SUBAPPLICATION Uebung_052_AX (* DigitalInput_I1-_I4 auf DigitalOutput_Q1-_Q4, mit Plug and Socket *)
  (* Standard: 61499-2; Description: Copyright (c) 2026 Meisterschulen am Ostbahnhof This program and the accompanying materials are made available under the terms of the Eclipse Public License 2.0 which is available at https://www.eclipse.org/legal/epl-2.0/ SPDX-License-Identifier: EPL-2.0 *)
  (* Version 1.0, 2026-09-09, Franz Höpfinger, Meisterschulen am Ostbahnhof, initial API and implementation and/or initial documentation *)
  PACKAGE Uebungen;
  IMPORT logiBUS::io::DI::logiBUS_DI::Input_I1;
  IMPORT logiBUS::io::DI::logiBUS_DI::Input_I2;
  IMPORT logiBUS::io::DI::logiBUS_DI::Input_I3;
  IMPORT logiBUS::io::DI::logiBUS_DI::Input_I4;
  IMPORT logiBUS::io::DQ::logiBUS_DO::Output_Q1;
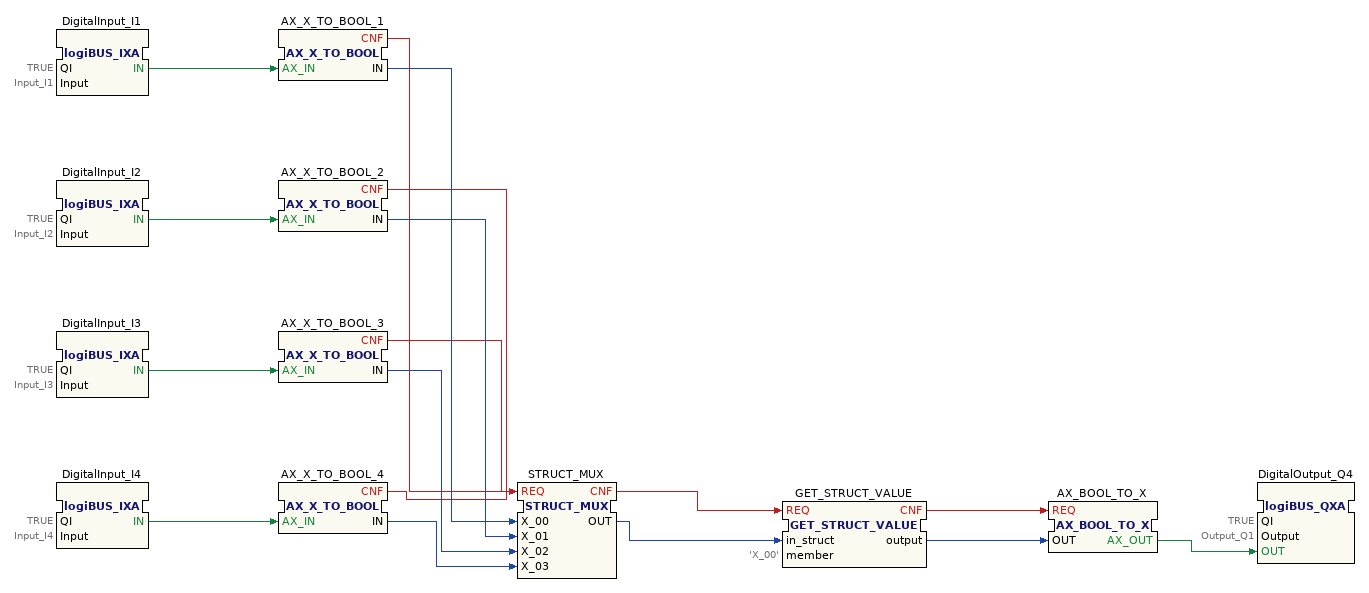
  FBS
    DigitalInput_I1 : logiBUS::io::DI::logiBUS_IXA(QI := TRUE, Input := Input_I1);
    DigitalInput_I2 : logiBUS::io::DI::logiBUS_IXA(QI := TRUE, Input := Input_I2);
    DigitalInput_I3 : logiBUS::io::DI::logiBUS_IXA(QI := TRUE, Input := Input_I3);
    DigitalOutput_Q4 : logiBUS::io::DQ::logiBUS_QXA(QI := TRUE, Output := Output_Q1);
    DigitalInput_I4 : logiBUS::io::DI::logiBUS_IXA(QI := TRUE, Input := Input_I4);
    GET_STRUCT_VALUE : eclipse4diac::convert::GET_STRUCT_VALUE(member := 'X_00');
    STRUCT_MUX : eclipse4diac::convert::STRUCT_MUX; {SET_ATTRIBUTE(StructuredType, logiBUS::utils::conversion::types::ST04X)}
    AX_X_TO_BOOL_1 : adapter::conversion::unidirectional::AX_X_TO_BOOL;
    AX_X_TO_BOOL_2 : adapter::conversion::unidirectional::AX_X_TO_BOOL;
    AX_X_TO_BOOL_3 : adapter::conversion::unidirectional::AX_X_TO_BOOL;
    AX_X_TO_BOOL_4 : adapter::conversion::unidirectional::AX_X_TO_BOOL;
    AX_BOOL_TO_X : adapter::conversion::unidirectional::AX_BOOL_TO_X;
  END_FBS
  EVENT_CONNECTIONS
    GET_STRUCT_VALUE.CNF TO AX_BOOL_TO_X.REQ;
    AX_X_TO_BOOL_1.CNF TO STRUCT_MUX.REQ;
    AX_X_TO_BOOL_2.CNF TO STRUCT_MUX.REQ;
    AX_X_TO_BOOL_3.CNF TO STRUCT_MUX.REQ;
    AX_X_TO_BOOL_4.CNF TO STRUCT_MUX.REQ;
    STRUCT_MUX.CNF TO GET_STRUCT_VALUE.REQ;
  END_CONNECTIONS
  DATA_CONNECTIONS
    GET_STRUCT_VALUE.output TO AX_BOOL_TO_X.OUT;
    AX_X_TO_BOOL_1.IN TO STRUCT_MUX.X_00;
    AX_X_TO_BOOL_2.IN TO STRUCT_MUX.X_01;
    AX_X_TO_BOOL_3.IN TO STRUCT_MUX.X_02;
    AX_X_TO_BOOL_4.IN TO STRUCT_MUX.X_03;
    STRUCT_MUX.OUT TO GET_STRUCT_VALUE.in_struct;
  END_CONNECTIONS
  ADAPTER_CONNECTIONS
    DigitalInput_I1.IN TO AX_X_TO_BOOL_1.AX_IN;
    DigitalInput_I2.IN TO AX_X_TO_BOOL_2.AX_IN;
    DigitalInput_I3.IN TO AX_X_TO_BOOL_3.AX_IN;
    DigitalInput_I4.IN TO AX_X_TO_BOOL_4.AX_IN;
    AX_BOOL_TO_X.AX_OUT TO DigitalOutput_Q4.OUT;
  END_CONNECTIONS
END_SUBAPPLICATION
